Yaskawa INFORM job: FRONT_SEARCH_90ST-1_5340.JBI

/JOB
//NAME FRONT_SEARCH_90ST-1_5340
///FOLDERNAME 02-SKRZYNIE_JOBS
//POS
///NPOS 44,44,0,8,0,0
///TOOL 0
///POSTYPE PULSE
///PULSE
C00000=0,-52278,40443,0,6873,1
C00001=-51470,-5720,51886,-842,-6167,45146
C00002=-68922,2266,43359,-60391,-17537,61768
C00003=-68922,2266,43359,-60391,-17537,61768
C00004=-68101,12166,56995,-54361,-18113,58924
C00005=-67210,13249,58456,-52695,-17792,58254
C00006=-68101,12166,56995,-54361,-18113,58924
C00007=-69177,13734,59118,-55068,-18794,59090
C00008=-57226,3834,46972,-36987,-12966,52270
C00009=-57226,5214,50337,-33908,-13993,50784
C00010=-57226,1690,41664,-43028,-11428,55171
C00011=-39195,-4952,37289,18918,-10992,28464
C00012=-62169,-6896,8508,43480,33664,19777
C00013=-60930,-5588,9811,42688,33146,20317
C00014=-61169,-5094,11915,43959,32492,19583
C00015=-62169,-6896,8508,43480,33664,19777
C00016=-15265,-21103,6084,128589,-10550,-14483
C00017=-15265,-21103,6084,128589,-10550,-14483
C00018=-14836,-19577,7234,129073,-10997,-14667
C00019=-14920,-18994,9366,125223,-10278,-12842
C00020=-15265,-21103,6084,128589,-10550,-14483
C00021=16867,-24115,-4728,128463,-25926,-4026
C00022=14148,-24463,-4976,130369,-24563,-5269
C00023=13812,-23136,-4020,131151,-24649,-5704
C00024=13890,-22573,-1750,129338,-23891,-4758
C00025=14148,-24463,-4976,130369,-24563,-5269
C00026=19623,-34877,-16768,124729,-29078,51940
C00027=17214,-25882,-2994,159745,-10910,31509
C00028=21601,-24733,-1135,146987,-11593,38051
C00029=20844,-22883,174,149935,-11807,36561
C00030=20964,-22504,1816,147814,-11082,37587
C00031=20152,-29372,-7837,152831,-12202,35107
C00032=58163,-16078,3541,118491,-24924,50999
C00033=57910,-10436,12617,114927,-23770,52815
C00034=56655,-9151,13822,115844,-23121,52219
C00035=57911,-10438,12617,114927,-23770,52814
C00036=57911,-9269,15925,112152,-23134,54238
C00037=50865,-11274,17469,103402,-13103,62071
C00038=52641,-10121,17568,107927,-14239,60207
C00039=55122,-10973,14720,110381,-19153,56434
C00040=46873,-31323,-15655,127144,-23194,47707
C00041=53252,-41973,-2905,102185,-37459,42403
C00042=0,-35574,42087,36666,-9339,1809
C00043=0,-52278,40443,0,6873,1
BC00000=863743
BC00001=949183
BC00002=1000773
BC00003=1000773
BC00004=1000773
BC00005=1000773
BC00006=1000773
BC00007=1000773
BC00008=1000774
BC00009=1000774
BC00010=1000774
BC00011=1000774
BC00012=1000774
BC00013=1000774
BC00014=1000774
BC00015=1000774
BC00016=1000774
BC00017=1000774
BC00018=1000774
BC00019=1000774
BC00020=1000774
BC00021=1000774
BC00022=1000774
BC00023=1000774
BC00024=1000774
BC00025=1000774
BC00026=1000774
BC00027=1000774
BC00028=1000774
BC00029=1000774
BC00030=1000774
BC00031=1000774
BC00032=1000771
BC00033=1000771
BC00034=1000772
BC00035=1000772
BC00036=1000772
BC00037=1000772
BC00038=1000772
BC00039=1000772
BC00040=1000772
BC00041=942070
BC00042=827719
BC00043=820842
///POSTYPE BASE
///RECTAN
///RCONF 1,0,0,0,0,0,0,0,0,0,0,0,0,0,0,0,0,0,0,0,0,0,0,0
P00006=0.000,0.000,0.000,0.0000,0.0000,0.0000
///RCONF 0,0,0,0,0,0,0,0,0,0,0,0,0,0,0,0,0,0,0,0,0,0,0,0
P00058=0.000,0.000,3.000,0.0000,0.0000,0.0000
///RCONF 1,0,0,0,0,0,0,0,0,0,0,0,0,0,0,0,0,0,0,0,0,0,0,0
P00500=2.332,-5.281,-1.258,0.0000,0.0000,0.0000
///RCONF 0,0,0,0,0,0,0,0,0,0,0,0,0,0,0,0,0,0,0,0,0,0,0,0
P00501=-2.026,0.009,3.534,0.0000,0.0000,0.0000
///RCONF 1,0,0,0,0,0,0,0,0,0,0,0,0,0,0,0,0,0,0,0,0,0,0,0
P00502=-2.023,0.001,1.732,0.0000,0.0000,0.0000
P00503=0.138,-0.044,1.539,0.0000,0.0000,0.0000
P00504=-0.309,-0.010,1.636,0.0000,0.0000,0.0000
P00505=0.999,-9.916,8.214,0.0000,0.0000,0.0000
//INST
///DATE 2024/08/01 15:51
///ATTR SC,RW
///GROUP1 RB1,BS1
NOP
MOVJ C00000 BC00000 VJ=50.00
MOVJ C00001 BC00001 VJ=50.00
MOVJ C00002 BC00002 VJ=30.00
'::::::::::::::::::::::::::::::::
'W21 P
'::::::::::::::::::::::::::::::::
MOVL C00003 BC00003 V=500.0
MOVL C00004 BC00004 V=333.3 PL=0
REFP 3 C00005 BC00005
CALL JOB:SEARCH-R1
SET P0500 P0006
SFTON P0500
MOVL C00006 BC00006 V=333.3 PL=0
REFP 3 C00007 BC00007
CALL JOB:SEARCH-R1
SET P0500 P0006
SFTON P0500
MOVL C00008 BC00008 V=333.3 PL=0
REFP 3 C00009 BC00009
CALL JOB:SEARCH-R1
SET P0500 P0006
SFTOF
MOVL C00010 BC00010 V=166.7
'::::::::::::::::::::::::::::::::
'W21 L
'::::::::::::::::::::::::::::::::
MOVL C00011 BC00011 V=333.3
MOVL C00012 BC00012 V=333.3 PL=0
REFP 3 C00013 BC00013
CALL JOB:SEARCH-R1
IMOV P0058 V=16.7
SET P0501 P0006
SFTON P0501
REFP 3 C00014 BC00014
CALL JOB:SEARCH-R1
SET P0501 P0006
SFTON P0501
MOVL C00015 BC00015 V=500.0 PL=0
SFTOF
'::::::::::::::::::::::::::::::::
'W20 P
'::::::::::::::::::::::::::::::::
MOVL C00016 BC00016 V=250.0
MOVL C00017 BC00017 V=333.3 PL=0
REFP 3 C00018 BC00018
CALL JOB:SEARCH-R1
IMOV P0058 V=16.7
SET P0502 P0006
SFTON P0502
REFP 3 C00019 BC00019
CALL JOB:SEARCH-R1
SET P0502 P0006
SFTON P0502
MOVL C00020 BC00020 V=500.0 PL=0
SFTOF
'::::::::::::::::::::::::::::::::
'W20 L
'::::::::::::::::::::::::::::::::
MOVL C00021 BC00021 V=250.0
MOVL C00022 BC00022 V=333.3 PL=0
REFP 3 C00023 BC00023
CALL JOB:SEARCH-R1
IMOV P0058 V=16.7
SET P0503 P0006
SFTON P0503
REFP 3 C00024 BC00024
CALL JOB:SEARCH-R1
SET P0503 P0006
SFTON P0503
MOVL C00025 BC00025 V=500.0 PL=0
SFTOF
'::::::::::::::::::::::::::::::::
'W22 P
'::::::::::::::::::::::::::::::::
MOVL C00026 BC00026 V=166.7
MOVL C00027 BC00027 V=333.3
MOVL C00028 BC00028 V=333.3 PL=0
REFP 3 C00029 BC00029
CALL JOB:SEARCH-R1
IMOV P0058 V=16.7
SET P0504 P0006
SFTON P0504
REFP 3 C00030 BC00030
CALL JOB:SEARCH-R1
SET P0504 P0006
SFTON P0504
MOVL C00031 BC00031 V=500.0 PL=0
SFTOF
'::::::::::::::::::::::::::::::::
'W22 L
'::::::::::::::::::::::::::::::::
MOVL C00032 BC00032 V=333.3
MOVL C00033 BC00033 V=333.3 PL=0
REFP 3 C00034 BC00034
CALL JOB:SEARCH-R1
SET P0505 P0006
SFTON P0505
MOVL C00035 BC00035 V=333.3 PL=0
REFP 3 C00036 BC00036
CALL JOB:SEARCH-R1
SET P0505 P0006
SFTON P0505
MOVL C00037 BC00037 V=333.3 PL=0
REFP 3 C00038 BC00038
CALL JOB:SEARCH-R1
SET P0505 P0006
SFTOF
MOVL C00039 BC00039 V=83.3
MOVL C00040 BC00040 V=333.3
MOVJ C00041 BC00041 VJ=40.00
MOVJ C00042 BC00042 VJ=80.00
MOVJ C00043 BC00043 VJ=80.00
END
